Staubli VAL3: readFileList.pgx

public program readFileList(string x_sFileFolder, string& x_sFileList[])
begin
  //读取robotmaster生成的全部文件列表
  resize(x_sFileList,1,1)
  x_sFileList[0]=""
  if !libList(x_sFileFolder,x_sFileList)
    logMsg("读取文件列表错误")
  endIf
end
